FUNCTION_BLOCK FB_Sensor_NO_2InRow_TestDecorator EXTENDS FB_Sensor_TestParentDecorator IMPLEMENTS ITF_Sensor_NO_2InRow_TestDecorator
VAR
	bContact2Test			: BOOL;
END_VAR

(*			
	EVERDE sp. z o.o.
	Rafał Osajda		05.02.2025		TC 4026.13		wer. 0.0.0.1
	Zwraca aktualny stan czujnika
*)
METHOD IsActive : BOOL
IsActive			:= THIS^.bContactTest AND THIS^.bContact2Test;
END_METHOD

METHOD PUBLIC SetContact2
VAR_INPUT
	bIN: BOOL;
END_VAR
THIS^.bContact2Test		:= bIN;
END_METHOD

END_FUNCTION_BLOCK

(* stored: Version 1.1.0.1
   POU FB_Sensor_NO_2InRow_TestDecorator: Id {b6fc94cc-8edf-4c59-ba2e-b635d54a6a05}, SpecialFunc None
   Method IsActive: Id {dc3a6181-5590-49f7-ba67-843aca16ce19}
   Method SetContact2: Id {84549dab-3535-4e89-a4be-6b43738e7357} *)
